Universal Robots PolyScope program: ctito_pp.urp

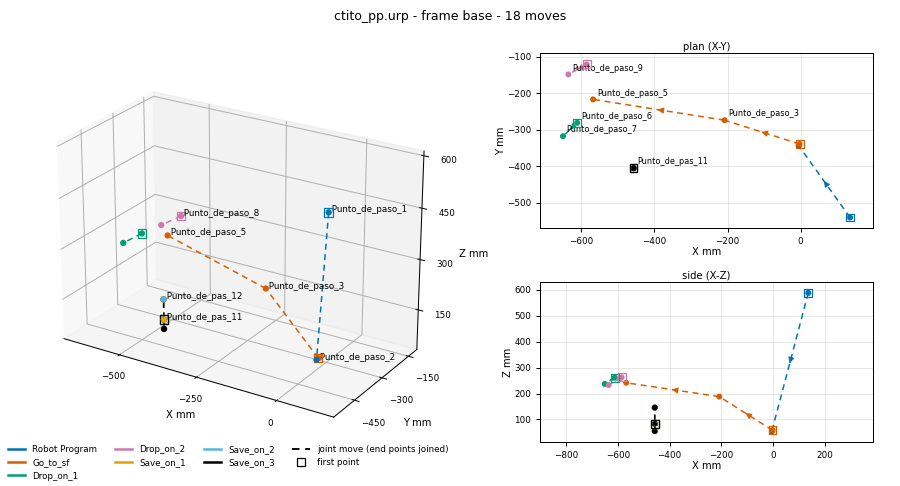
[picture p0: tool path of ctito_pp.urp in frame base, 18 of 18 moves have a stored position in this frame; points joined in program order, loops and branches not executed]
Program ctito_pp (installation=default directory=/home/ur/ursim-current/programs/Clasificador TITO/ctito_pp createdIn=3.5.3.10825 lastSavedIn=3.12.1.90940 robotSerialNumber=2018359999)
Calibrated DH parameters: a=[0, -0.425, -0.39225, 0, 0, 0]; d=[0.089159, 0, 0, 0.10915, 0.09465, 0.0823]; alpha=[1.570796, 0, 0, 1.570796, -1.570796, 0]; deltaTheta=[0, 0, 0, 0, 0, 0]
Robot Program (runOnlyOnce=false)
  MoveJ speed 60 deg/s, acceleration 80 deg/s^2 (useActiveTCP=false)
    Waypoint Punto_de_paso_1: TCP in base x=135.062 y=-539.888 z=588.326 mm, rx=-0.0336 ry=2.1619 rz=-2.0853 rad; joints [89.322, -105.154, 104.809, -177.851, -82.761, 4.553] deg; flange x=115.187 y=-367.114 z=593.772 mm, rx=-0.0337 ry=2.1618 rz=-2.0853 rad
    SuppressedNode (comment=Gripper disabled (Only for sim))
      URCap Gripper (Robotiq_Grippers, Robotiq Inc.) dataModel(position=0.0, force=100.0, speed=100.0, positionInDouble=0.0, forceInDouble=100.0, speedInDouble=100.0, slaveIds=[9], blocking=true)
    If cont_process≟3
      Popup Warning (haltProgram=false message=The output cups is over. inputType=Text)
      cont_process := 0
    If digital_in[0]
      Popup Message (haltProgram=false message=Has been detected a cup inputType=Text)
      Waypoint Punto_de_paso_2: TCP in base x=-5.432 y=-343.453 z=54.78 mm, rx=-0.0837 ry=2.3833 rz=2.0448 rad; joints [79.785, -52.289, 89.643, -46.331, -102.068, -3.915] deg; flange x=0.564 y=-515.304 z=81.336 mm, rx=-0.0837 ry=2.3832 rz=2.0448 rad
      SuppressedNode
        URCap Gripper (Robotiq_Grippers, Robotiq Inc.) dataModel(position=9.362181654270898, force=100.0, speed=100.0, positionInDouble=9.362181654270898, forceInDouble=100.0, speedInDouble=100.0, slaveIds=[9], blocking=true); state(isChildrenLocked=true)
      Call Go_to_sf
      If (digital_in[1] and digital_in[2]) or ( not digital_in[1] and digital_in[3])
        Call Drop_on_1
      Else 
        Call Drop_on_2
      SuppressedNode
        Waypoint Punto_de_pas_11: TCP in base x=-457.215 y=-404.963 z=83.7 mm, rx=1.6972 ry=0.1493 rz=0.0246 rad; joints [5.046, -43.349, 87.778, 52.459, 7.673, -101.031] deg; flange x=-475.193 y=-233.417 z=106.75 mm, rx=1.6973 ry=0.1493 rz=0.0246 rad
      SuppressedNode
        Waypoint Punto_de_pas_10: TCP in base x=-457.269 y=-404.933 z=55.133 mm, rx=1.6971 ry=0.1494 rz=0.0244 rad; joints [5.046, -40.581, 87.806, 49.663, 7.673, -101.031] deg; flange x=-475.193 y=-233.417 z=78.154 mm, rx=1.6973 ry=0.1493 rz=0.0246 rad
      SuppressedNode
        URCap Gripper (Robotiq_Grippers, Robotiq Inc.) dataModel(position=0.0, force=100.0, speed=100.0, positionInDouble=0.0, forceInDouble=100.0, speedInDouble=100.0, slaveIds=[9], blocking=true); state(isChildrenLocked=true)
      SuppressedNode
        Waypoint Punto_de_pas_12: TCP in base x=-457.267 y=-404.928 z=145.856 mm, rx=1.6973 ry=0.1492 rz=0.0247 rad; joints [5.046, -48.875, 86.745, 59.017, 7.673, -101.031] deg; flange x=-475.193 y=-233.417 z=168.945 mm, rx=1.6973 ry=0.1493 rz=0.0246 rad
      Switch expression=cont_process
        Case (caseValue=0)
          Call Save_on_1
        Case (caseValue=1)
          Call Save_on_2
        Case (caseValue=2)
          Call Save_on_3
      Set IncrementVariable installationVariable=cont_process
SubProgram -> Go_to_sf
SubProgram -> Drop_on_1
SubProgram -> Drop_on_2
SubProgram -> Save_on_1
SubProgram -> Save_on_2
SubProgram -> Save_on_3
SubProgram Go_to_sf (keepSynchronizedWithDisk=false)
  MoveJ speed 60 deg/s, acceleration 80 deg/s^2 (useActiveTCP=true)
    Waypoint Punto_de_paso_4: TCP in base x=-2.786 y=-338.929 z=58.485 mm, rx=0.0777 ry=-2.4498 rz=-1.9359 rad; joints [80.163, -55.861, 91.967, -49.805, -102.155, -3.913] deg; flange x=5.101 y=-508.011 z=98.765 mm, rx=0.0778 ry=-2.4497 rz=-1.936 rad
    Waypoint Punto_de_paso_3: TCP in base x=-208.206 y=-273.817 z=188.244 mm, rx=1.0691 ry=1.9893 rz=1.171 rad; joints [31.634, -71.953, 87.837, -42.01, -86.696, -3.914] deg; flange x=-346.265 y=-347.072 z=264.736 mm, rx=1.0692 ry=1.9893 rz=1.171 rad
    Waypoint Punto_de_paso_5: TCP in base x=-567.711 y=-216.824 z=241.713 mm, rx=1.5944 ry=-0.1577 rz=0.0724 rad; joints [-15.349, -67.27, 87.849, -28.772, -12.497, 16.323] deg; flange x=-558.65 y=-43.171 z=247.054 mm, rx=1.5943 ry=-0.1577 rz=0.0725 rad
SubProgram Drop_on_1 (keepSynchronizedWithDisk=false)
  MoveJ speed 60 deg/s, acceleration 80 deg/s^2 (useActiveTCP=true)
    Waypoint Punto_de_paso_6: TCP in base x=-611.435 y=-280.889 z=261.641 mm, rx=1.554 ry=-0.2446 rz=0.2303 rad; joints [-8.003, -58.645, 72.876, -13.197, -7.463, 16.325] deg; flange x=-609.783 y=-106.897 z=261.218 mm, rx=1.5539 ry=-0.2446 rz=0.2305 rad
    Waypoint Punto_de_paso_7: TCP in base x=-650.23 y=-317.539 z=237.272 mm, rx=0.9145 ry=-1.5222 rz=1.4392 rad; joints [-4.301, -55.884, 72.109, -20.339, 0.622, 117.205] deg; flange x=-635.284 y=-144.204 z=237.081 mm, rx=0.9144 ry=-1.5222 rz=1.4393 rad
SubProgram Drop_on_2 (keepSynchronizedWithDisk=false)
  MoveJ speed 60 deg/s, acceleration 80 deg/s^2 (useActiveTCP=true)
    Waypoint Punto_de_paso_8: TCP in base x=-585.345 y=-121.081 z=262.635 mm, rx=1.5558 ry=-0.2067 rz=0.2651 rad; joints [-23.106, -58.599, 72.851, -13.249, -25.191, 16.317] deg; flange x=-591.672 y=52.808 z=261.32 mm, rx=1.5557 ry=-0.2068 rz=0.2651 rad
    Waypoint Punto_de_paso_9: TCP in base x=-635.382 y=-148.533 z=233.099 mm, rx=0.9579 ry=-1.5407 rz=1.4944 rad; joints [-19.563, -54.605, 70.016, -18.095, -18.152, 117.388] deg; flange x=-631.051 y=25.416 z=235.625 mm, rx=0.9578 ry=-1.5408 rz=1.4944 rad
SubProgram Save_on_1 (keepSynchronizedWithDisk=false)
  MoveJ speed 60 deg/s, acceleration 80 deg/s^2 (useActiveTCP=true)
    Waypoint Punto_de_pas_11: TCP in base x=-457.215 y=-404.963 z=83.7 mm, rx=1.6972 ry=0.1493 rz=0.0246 rad; joints [5.046, -43.349, 87.778, 52.459, 7.673, -101.031] deg; flange x=-475.193 y=-233.417 z=106.75 mm, rx=1.6973 ry=0.1493 rz=0.0246 rad
    Waypoint Punto_de_pas_10: TCP in base x=-457.269 y=-404.933 z=55.133 mm, rx=1.6971 ry=0.1494 rz=0.0244 rad; joints [5.046, -40.581, 87.806, 49.663, 7.673, -101.031] deg; flange x=-475.193 y=-233.417 z=78.154 mm, rx=1.6973 ry=0.1493 rz=0.0246 rad
    Waypoint Punto_de_pas_12: TCP in base x=-457.267 y=-404.928 z=145.856 mm, rx=1.6973 ry=0.1492 rz=0.0247 rad; joints [5.046, -48.875, 86.745, 59.017, 7.673, -101.031] deg; flange x=-475.193 y=-233.417 z=168.945 mm, rx=1.6973 ry=0.1493 rz=0.0246 rad
SubProgram Save_on_2 (keepSynchronizedWithDisk=false)
  MoveJ speed 60 deg/s, acceleration 80 deg/s^2 (useActiveTCP=true)
    Waypoint Punto_de_pas_11: TCP in base x=-457.215 y=-404.963 z=83.7 mm, rx=1.6972 ry=0.1493 rz=0.0246 rad; joints [5.046, -43.349, 87.778, 52.459, 7.673, -101.031] deg; flange x=-475.193 y=-233.417 z=106.75 mm, rx=1.6973 ry=0.1493 rz=0.0246 rad
    Waypoint Punto_de_pas_10: TCP in base x=-457.269 y=-404.933 z=55.133 mm, rx=1.6971 ry=0.1494 rz=0.0244 rad; joints [5.046, -40.581, 87.806, 49.663, 7.673, -101.031] deg; flange x=-475.193 y=-233.417 z=78.154 mm, rx=1.6973 ry=0.1493 rz=0.0246 rad
    Waypoint Punto_de_pas_12: TCP in base x=-457.267 y=-404.928 z=145.856 mm, rx=1.6973 ry=0.1492 rz=0.0247 rad; joints [5.046, -48.875, 86.745, 59.017, 7.673, -101.031] deg; flange x=-475.193 y=-233.417 z=168.945 mm, rx=1.6973 ry=0.1493 rz=0.0246 rad
SubProgram Save_on_3 (keepSynchronizedWithDisk=false)
  MoveJ speed 60 deg/s, acceleration 80 deg/s^2 (useActiveTCP=true)
    Waypoint Punto_de_pas_11: TCP in base x=-457.215 y=-404.963 z=83.7 mm, rx=1.6972 ry=0.1493 rz=0.0246 rad; joints [5.046, -43.349, 87.778, 52.459, 7.673, -101.031] deg; flange x=-475.193 y=-233.417 z=106.75 mm, rx=1.6973 ry=0.1493 rz=0.0246 rad
    Waypoint Punto_de_pas_10: TCP in base x=-457.269 y=-404.933 z=55.133 mm, rx=1.6971 ry=0.1494 rz=0.0244 rad; joints [5.046, -40.581, 87.806, 49.663, 7.673, -101.031] deg; flange x=-475.193 y=-233.417 z=78.154 mm, rx=1.6973 ry=0.1493 rz=0.0246 rad
    Waypoint Punto_de_pas_12: TCP in base x=-457.267 y=-404.928 z=145.856 mm, rx=1.6973 ry=0.1492 rz=0.0247 rad; joints [5.046, -48.875, 86.745, 59.017, 7.673, -101.031] deg; flange x=-475.193 y=-233.417 z=168.945 mm, rx=1.6973 ry=0.1493 rz=0.0246 rad
